{attribute 'GeneratedUsingTerminal: EL3051-0000-0016'}
{attribute addProperty BoxType "EL3051-0000-0016"}
{attribute addProperty Description "EL3051 1Ch. Ana. Input 4-20mA"}
{attribute addProperty Physics "KK"}
{attribute addProperty Id "AI_StandardAT %I*AI_Standard_EA9DF21E9WcStateAT %I*WcState_9091E0EB2InfoDataAT %I*InfoData_32EB74EA10"}
{attribute addProperty CRC "1765360954"}
{attribute addProperty Size "21"}
TYPE EL3051_6939453A EXTENDS EtcSlaveTerminalBase_947E5A46 :
STRUCT
	{attribute addProperty Name "AI_Standard"}
	AI_Standard : AI_Standard_EA9DF21E;
	{attribute addProperty Name "WcState"}
	WcState : WcState_9091E0EB;
	{attribute addProperty Name "InfoData"}
	InfoData : InfoData_32EB74EA;
END_STRUCT
END_TYPE

(* stored: Version 1.2.0.0, ProductVersion 3.1.4024.9
   DUT EL3051_6939453A: Id {c6540c0a-f8df-4cdf-8723-a438280a444d} *)
